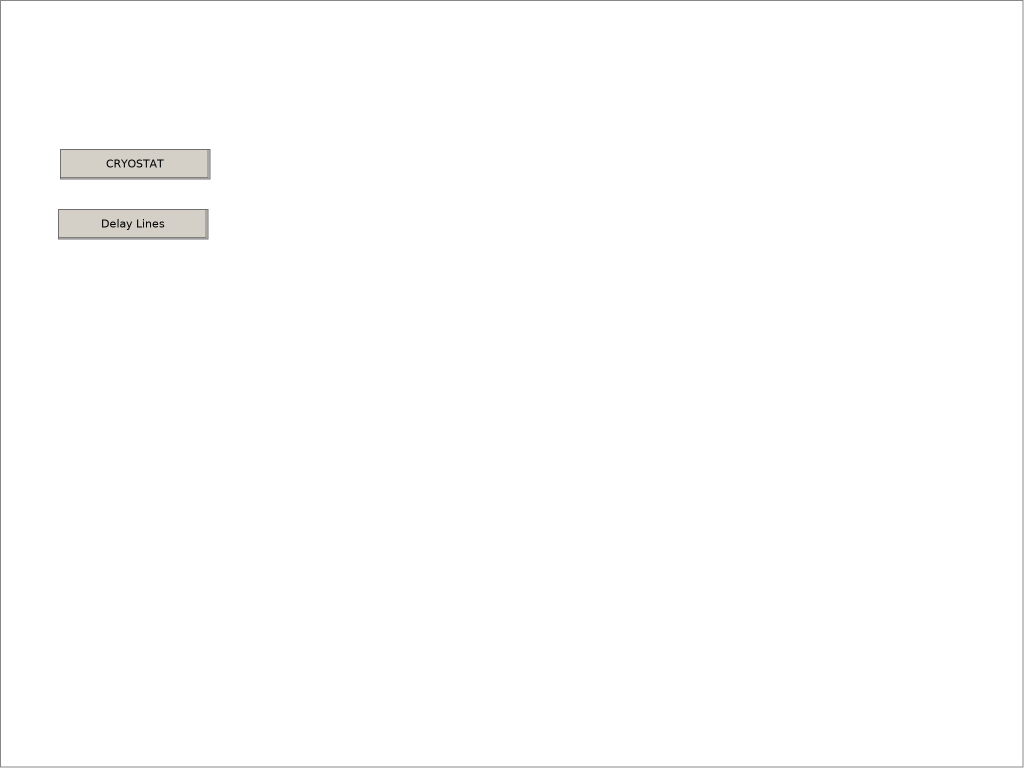
VISUALIZATION SCIFY_main  // 1024x768
    Button (60,149 150x30), "CRYOSTAT"
        OnMouseDown: change screen: SCIFY_Cryo
    Button (58,209 150x30), "Delay Lines"
        OnMouseDown: change screen: SCIFY_Delay_Lines
END_VISUALIZATION

(* stored: Version 1.1.0.1, ProductVersion 3.1.4024.12
   Visu SCIFY_main: Id {0ecbbf72-3d1d-47ab-bb9e-c12829a757ff} *)
